// Mitsubishi GX Works2 project: PID_slave_test1   PLC: FX3U/FX3UC

// global labels: Global1
VAR_GLOBAL
  lampe_0 AT Y000 : BOOL;
  lampe_1 AT Y001 : BOOL;
  lampeVar_0 AT M100 : BOOL;
  lampeVar_1 AT M101 : BOOL;
  anaDig AT D8260 : INT;
  digAna AT D8262 : INT;
  slider AT D0 : INT;
  tank AT D1 : INT;
  Output_PID AT D40 : INT;  (* Utgangs signal sendt ut fra PID *)
  Input_Referance AT D42 : INT;  (* Referanse verdi sendt til PID *)
  Input_Process AT D44 : INT;  (* Prosess verdi Sendt til PID *)
  Input_ManualValue AT D54 : INT;  (* Manuell verdi sendt til PID *)
  Input_ManualMode AT M105 : BOOL;  (* Valg av Manuell "1" eller Auto "0" *)
  Input_SamplingsTime AT D56 : INT;  (* Samplingstid sendt til PID *)
  Input_OperationModus AT M106 : BOOL;  (* Valg av direkte "1" eller Revers "0" Regulering *)
  Inpud_IntegratorModus AT M107 : BOOL;  (* Valg av Integrator virkning på regulator *)
  Input_NomValue AT D58 : INT;  (* Nominelt pådrag *)
  Input_DerivatorModus AT M108 : BOOL;  (* Valg av Derivator virkning på regulator *)
  Input_MaxPådrag AT D60 : INT;  (* Max pådrag *)
  Input_MinPådrag AT D62 : INT;  (* Min pådrag *)
END_VAR

// task Task_01 (event TRUE, interval 0, priority 31): POU_01

PROGRAM POU_01
VAR
  TestBlock_1 : TestBlock;
  tiss_1 : tiss;
  TestBlock_2 : TestBlock;
  tiss_2 : tiss;
  tiss_3 : tiss;
END_VAR
(* structured ladder/FBD written out as ST: instructions are called as NAME(EN, inputs, outputs); _pN, _eN, _tN stand for wires *)
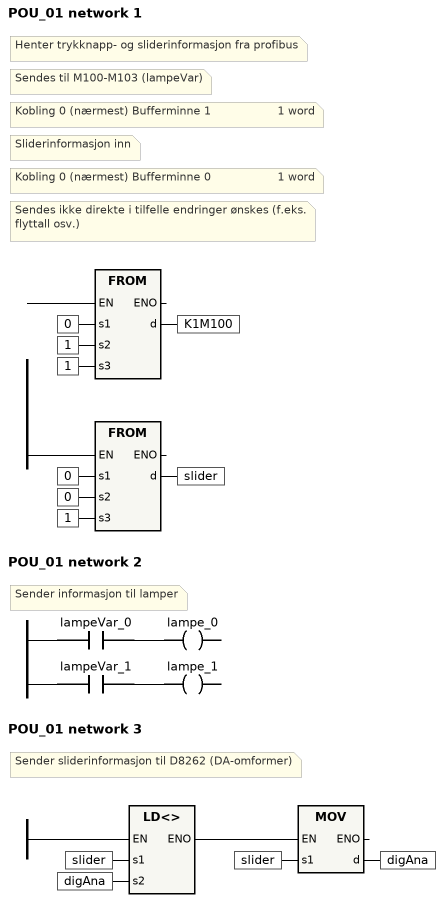
(* network 1 *)
(* Henter trykknapp- og sliderinformasjon fra profibus *)
(* Sendes til M100-M103 (lampeVar) *)
(* Kobling 0 (nærmest) Bufferminne 1                   1 word *)
(* Sliderinformasjon inn *)
(* Kobling 0 (nærmest) Bufferminne 0                   1 word *)
(* Sendes ikke direkte i tilfelle endringer ønskes (f.eks. flyttall osv.) *)
FROM(TRUE, 0, 1, 1, K1M100);
FROM(TRUE, 0, 0, 1, slider);
(* network 2 *)
(* Sender informasjon til lamper *)
lampe_0 := lampeVar_0;
lampe_1 := lampeVar_1;
(* network 3 *)
(* Sender sliderinformasjon til D8262 (DA-omformer) *)
_e1 := LD<>(TRUE, slider, digAna);
MOV(_e1, slider, digAna);
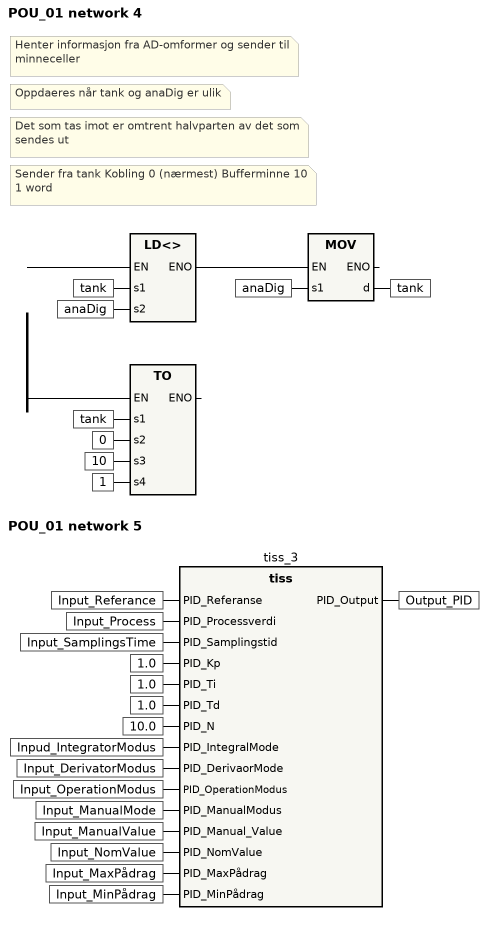
(* network 4 *)
(* Henter informasjon fra AD-omformer og sender til minneceller *)
(* Oppdaeres når tank og anaDig er ulik *)
(* Det som tas imot er omtrent halvparten av det som sendes ut *)
(* Sender fra tank Kobling 0 (nærmest) Bufferminne 10           1 word *)
_e1 := LD<>(TRUE, tank, anaDig);
MOV(_e1, anaDig, tank);
TO(TRUE, tank, 0, 10, 1);
(* network 5 *)
tiss_3(PID_Referanse := Input_Referance, PID_Processverdi := Input_Process, PID_Samplingstid := Input_SamplingsTime, PID_Kp := 1.0, PID_Ti := 1.0, PID_Td := 1.0, PID_N := 10.0, PID_IntegralMode := Inpud_IntegratorModus, PID_DerivaorMode := Input_DerivatorModus, PID_OperationModus := Input_OperationModus, PID_ManualModus := Input_ManualMode, PID_Manual_Value := Input_ManualValue, PID_NomValue := Input_NomValue, PID_MaxPådrag := Input_MaxPådrag, PID_MinPådrag := Input_MinPådrag, PID_Output => Output_PID);
END_PROGRAM

FUNCTION_BLOCK TestBlock
VAR_INPUT
  PID_Referanse : INT;  (* Referanseverdi PID blokk *)
  PID_Processverdi : INT;  (* Prosessverdi PID blokk *)
  PID_Samplingstid : REAL;  (* Samplingstid PID blokk (ms) *)
  PID_Kp : REAL;  (* KP PID blokk *)
  PID_Ti : REAL;  (* Ti PID blokk *)
  PID_Td : REAL;  (* Td PID blokk *)
  PID_N : REAL;  (* Filter konstant for Tf *)
  PID_IntegralMode : BOOL;  (* Integrator for PID blokk *)
  PID_DerivaorMode : BOOL;  (* Derivator for PID blokk *)
  PID_OperationModus : BOOL;  (* Framover kobling "0", bakoverkobling "1" *)
  PID_ManualModus : BOOL;  (* Auto "0" , Manuell pådrag "1" *)
END_VAR
VAR
  PID_Mellomregning_TN_F : REAL;  (* Mellomregning for T*N *)
  PID_Alpha : REAL;  (* Beregnet alpha verdi *)
  PID_ErrorValue_W : INT;  (* Beregnet error verdi *)
  PID_ErrorValue_F : ARRAY [0..1] OF REAL;  (* Beregnet error verdi *)
  PID_PGain : ARRAY [0..1] OF REAL;  (* Beregnet P forsterkning (Denne og forrige verdi) *)
  PID_Skalert_Processverdi_DW : DWORD;  (* Process verdi skalert med en faktor 2 *)
  PID_Skalert_Processverdi_W : WORD;  (* Process verdi skalert med en faktor 2 *)
  PID_Beta : REAL;  (* Beregnet alpha verdi *)
  PID_Mellomregning_TNplusTd_F : REAL;  (* Mellom regning for T*N+Td *)
  PID_Mellomregning_Integrator : REAL;  (* Mellom regning Kp*alpha*error[0] *)
  PID_IGain : ARRAY [0..1] OF REAL;  (* Beregnet I forsterkning (Denne og forrige verdi) *)
  PID_Mellomregning_Derivator : REAL;  (* Mellom regning for (Kp*Td/T)*(1-beta) *)
  PID_DGain : ARRAY [0..1] OF REAL;  (* Beregnet D forsterkning (Denne og forrige verdi) *)
  PID_Skalert_Processverdi_F : ARRAY [0..1] OF REAL;  (* Process verdi skalert med en faktor 2 *)
  PID_Gain : REAL;  (* Beregnet sum av pådrag *)
END_VAR
VAR_OUTPUT
  PID_Output : REAL;  (* Utgangsverdi fra PID-reg *)
END_VAR
(* structured ladder/FBD written out as ST: instructions are called as NAME(EN, inputs, outputs); _pN, _eN, _tN stand for wires *)
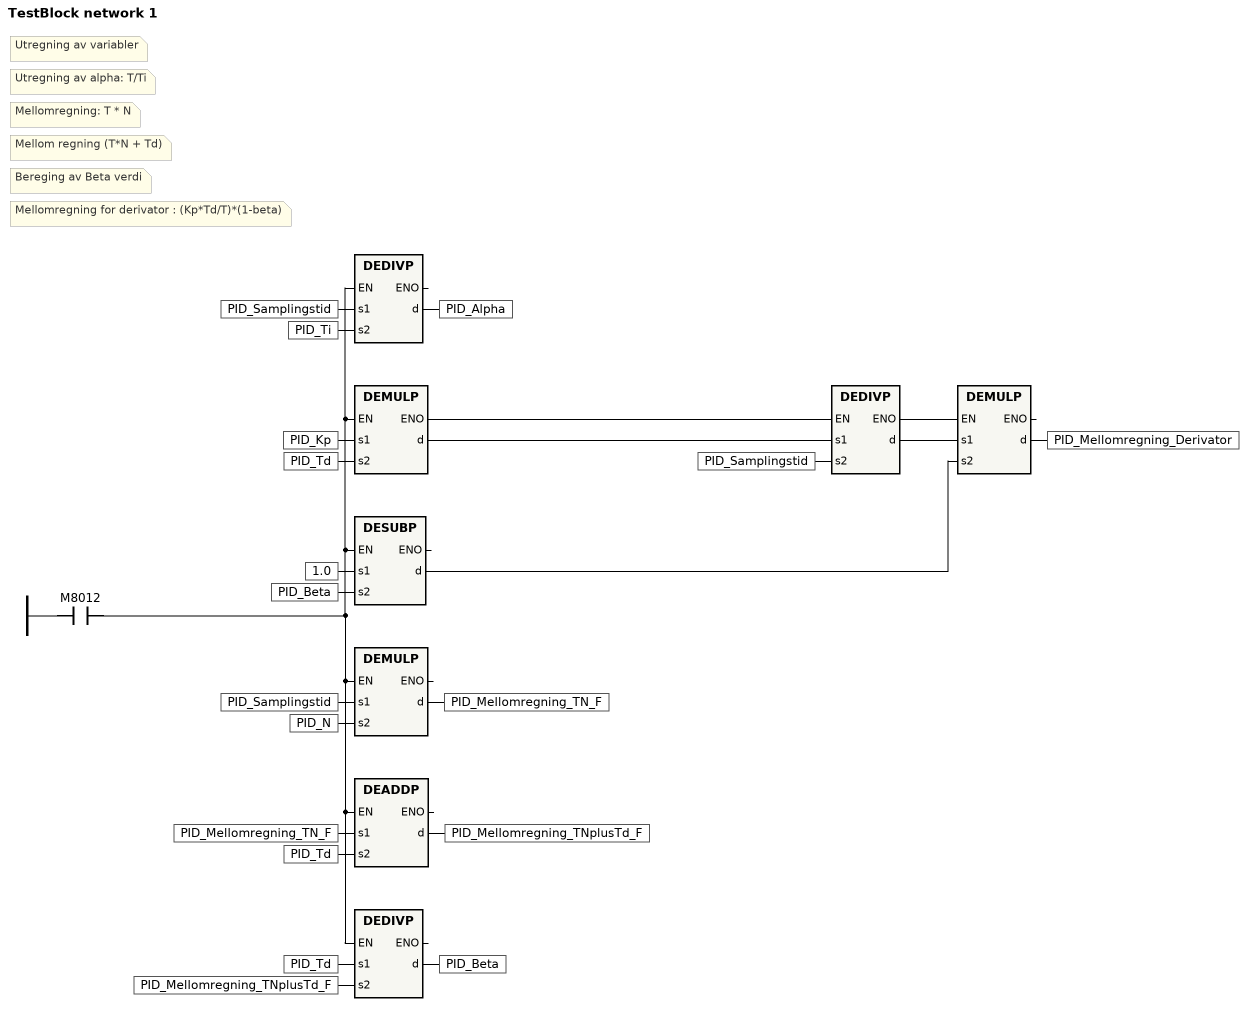
(* network 1 *)
(* Utregning av variabler *)
(* Utregning av alpha: T/Ti *)
(* Mellomregning: T * N *)
(* Mellom regning (T*N + Td) *)
(* Bereging av Beta verdi *)
(* Mellomregning for derivator : (Kp*Td/T)*(1-beta) *)
DEDIVP(M8012, PID_Samplingstid, PID_Ti, PID_Alpha);
DEMULP(M8012, PID_Samplingstid, PID_N, PID_Mellomregning_TN_F);
DEADDP(M8012, PID_Mellomregning_TN_F, PID_Td, PID_Mellomregning_TNplusTd_F);
DEDIVP(M8012, PID_Td, PID_Mellomregning_TNplusTd_F, PID_Beta);
_e2 := DEMULP(M8012, PID_Kp, PID_Td, _t1);
_e4 := DEDIVP(_e2, _t1, PID_Samplingstid, _t3);
DESUBP(M8012, 1.0, PID_Beta, _t5);
DEMULP(_e4, _t3, _t5, PID_Mellomregning_Derivator);
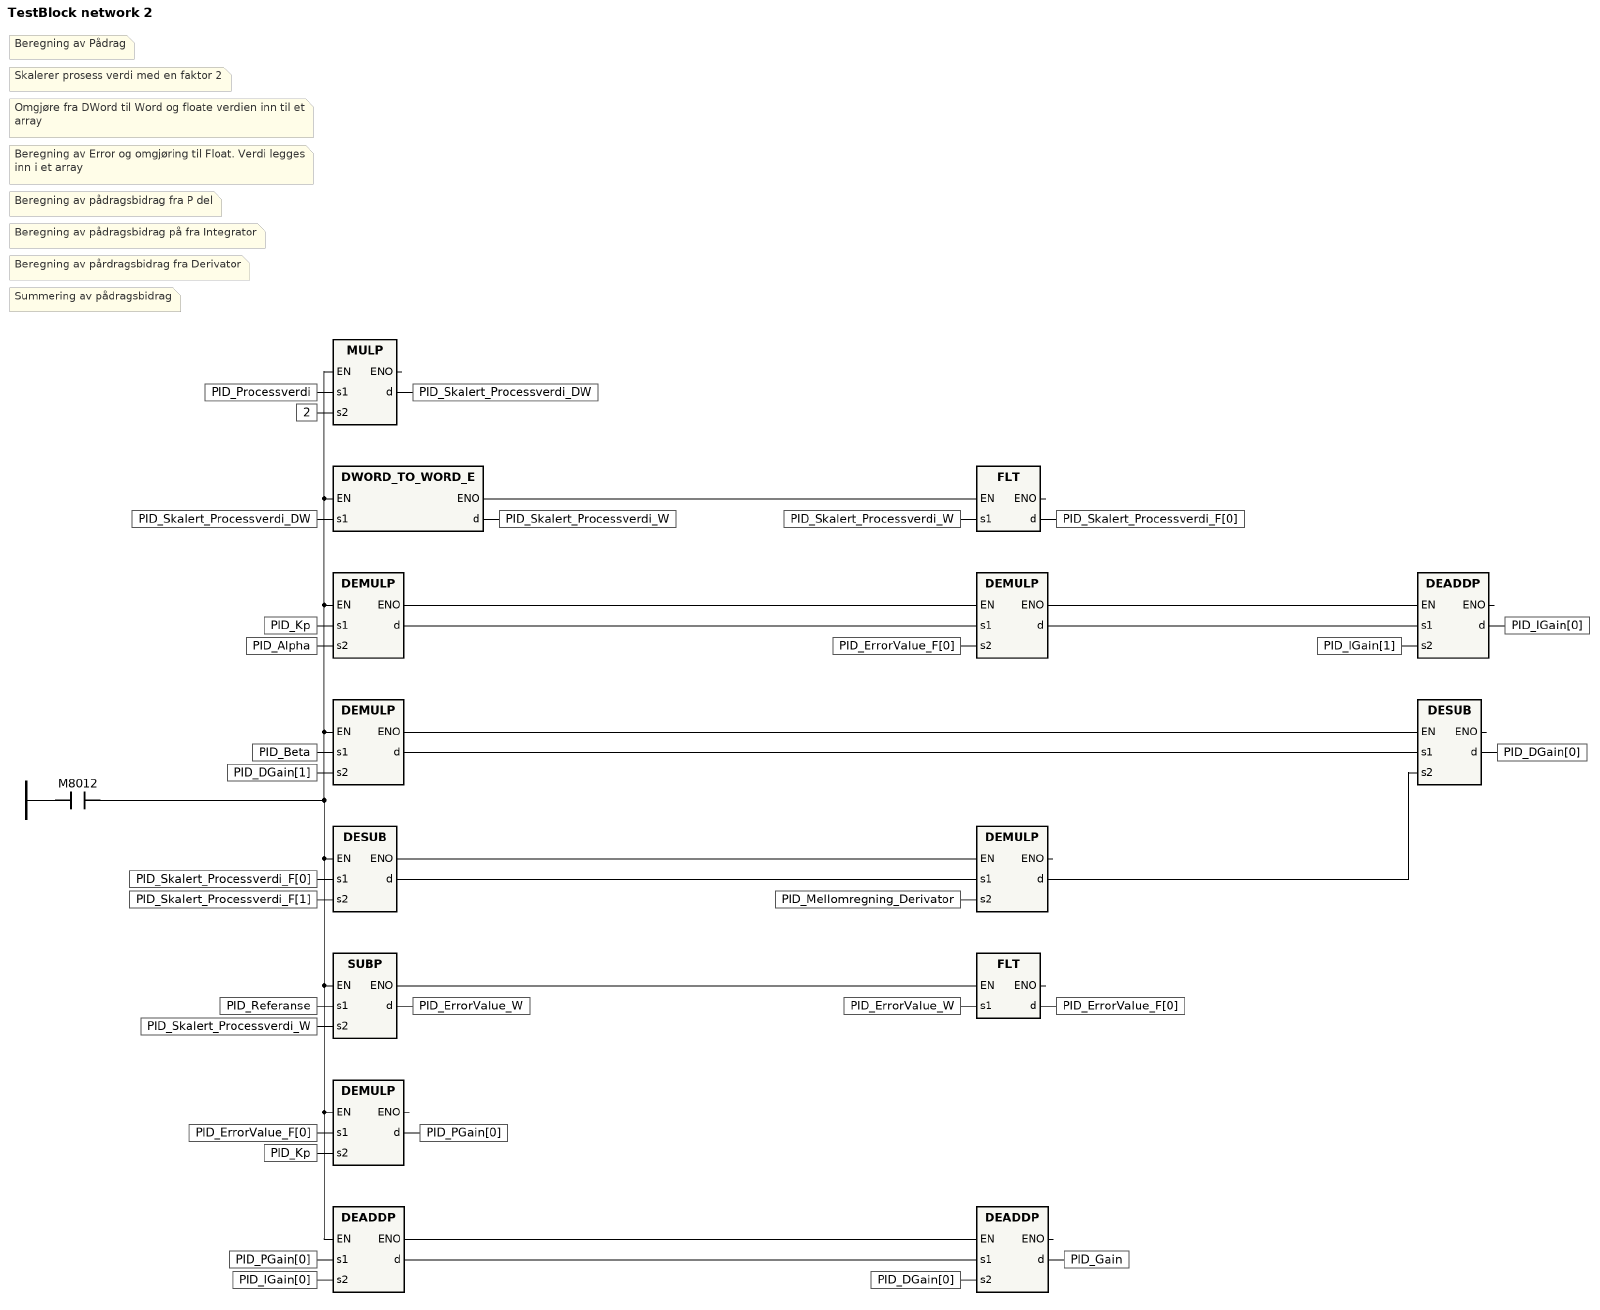
(* network 2 *)
(* Beregning av Pådrag *)
(* Skalerer prosess verdi med en faktor 2 *)
(* Omgjøre fra DWord til Word og floate verdien inn til et array *)
(* Beregning av Error og omgjøring til Float. Verdi legges inn i et array *)
(* Beregning av pådragsbidrag fra P del *)
(* Beregning av pådragsbidrag på fra Integrator *)
(* Beregning av pårdragsbidrag fra Derivator *)
(* Summering av pådragsbidrag *)
MULP(M8012, PID_Processverdi, 2, PID_Skalert_Processverdi_DW);
_e1 := DWORD_TO_WORD_E(M8012, PID_Skalert_Processverdi_DW, PID_Skalert_Processverdi_W);
FLT(_e1, PID_Skalert_Processverdi_W, PID_Skalert_Processverdi_F[0]);
_e2 := SUBP(M8012, PID_Referanse, PID_Skalert_Processverdi_W, PID_ErrorValue_W);
FLT(_e2, PID_ErrorValue_W, PID_ErrorValue_F[0]);
DEMULP(M8012, PID_ErrorValue_F[0], PID_Kp, PID_PGain[0]);
_e4 := DEMULP(M8012, PID_Kp, PID_Alpha, _t3);
_e6 := DEMULP(_e4, _t3, PID_ErrorValue_F[0], _t5);
DEADDP(_e6, _t5, PID_IGain[1], PID_IGain[0]);
_e8 := DEMULP(M8012, PID_Beta, PID_DGain[1], _t7);
_e10 := DESUB(M8012, PID_Skalert_Processverdi_F[0], PID_Skalert_Processverdi_F[1], _t9);
DEMULP(_e10, _t9, PID_Mellomregning_Derivator, _t11);
DESUB(_e8, _t7, _t11, PID_DGain[0]);
_e13 := DEADDP(M8012, PID_PGain[0], PID_IGain[0], _t12);
DEADDP(_e13, _t12, PID_DGain[0], PID_Gain);
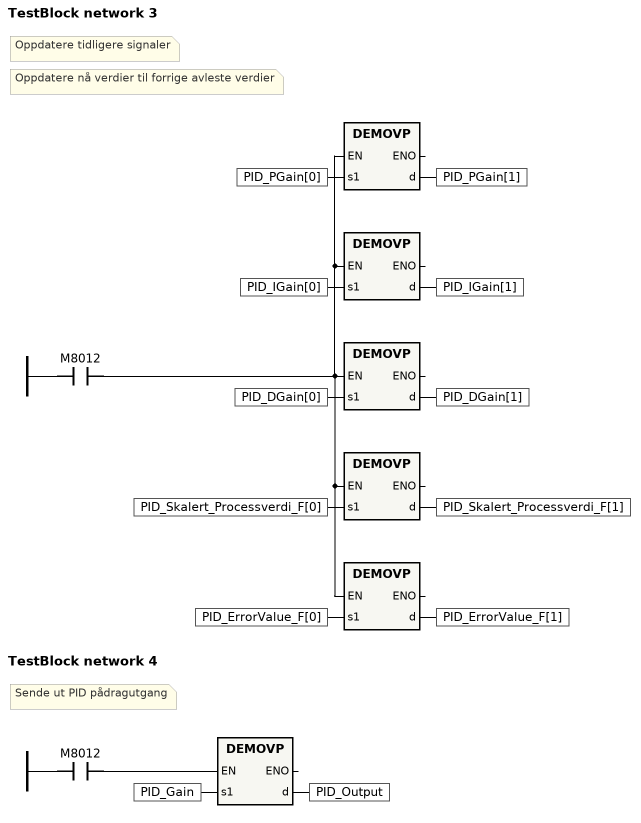
(* network 3 *)
(* Oppdatere tidligere signaler *)
(* Oppdatere nå verdier til forrige avleste verdier *)
DEMOVP(M8012, PID_PGain[0], PID_PGain[1]);
DEMOVP(M8012, PID_IGain[0], PID_IGain[1]);
DEMOVP(M8012, PID_DGain[0], PID_DGain[1]);
DEMOVP(M8012, PID_Skalert_Processverdi_F[0], PID_Skalert_Processverdi_F[1]);
DEMOVP(M8012, PID_ErrorValue_F[0], PID_ErrorValue_F[1]);
(* network 4 *)
(* Sende ut PID pådragutgang *)
DEMOVP(M8012, PID_Gain, PID_Output);
END_FUNCTION_BLOCK

FUNCTION_BLOCK tiss
VAR_INPUT
  PID_Referanse : INT;  (* Referanseverdi PID blokk *)
  PID_Processverdi : INT;  (* Prosessverdi PID blokk *)
  PID_Samplingstid : INT;  (* Samplingstid PID blokk (ms) *)
  PID_Kp : REAL;  (* KP PID blokk *)
  PID_Ti : REAL;  (* Ti PID blokk *)
  PID_Td : REAL;  (* Td PID blokk *)
  PID_N : REAL;  (* Filter konstant for Tf *)
  PID_IntegralMode : BOOL;  (* Integrator for PID blokk *)
  PID_DerivaorMode : BOOL;  (* Derivator for PID blokks *)
  PID_OperationModus : BOOL;  (* Direkte kobling "1", reversert "0" *)
  PID_ManualModus : BOOL;  (* Auto "0" , Manuell pådrag "1" *)
END_VAR
VAR
  PID_Alpha : REAL;  (* Beregnet alpha verdi *)
  PID_Beta : REAL;  (* Beregnet alpha verdi *)
END_VAR
VAR_INPUT
  PID_Manual_Value : INT;  (* Manuelt pådrag verdi *)
  PID_NomValue : INT;  (* Nominelt pådrags verdi *)
END_VAR
VAR_OUTPUT
  PID_Output : INT;  (* Utgangsverdi fra PID-reg *)
END_VAR
VAR_INPUT
  PID_MaxPådrag : INT;  (* Max pådrags verdi *)
  PID_MinPådrag : INT;  (* Min pådrags verdi *)
END_VAR
VAR
  PID_ErrorValue_F : ARRAY [0..1] OF REAL;  (* Beregnet error verdi *)
  PID_PGain : ARRAY [0..1] OF REAL;  (* Beregnet P forsterkning (Denne og forrige verdi) *)
  PID_IGain : ARRAY [0..1] OF REAL;  (* Beregnet I forsterkning (Denne og forrige verdi) *)
  PID_DGain : ARRAY [0..1] OF REAL;  (* Beregnet D forsterkning (Denne og forrige verdi) *)
  PID_Gain : REAL;  (* Beregnet sum av pådrag *)
  PID_Mellomregning_Samplingstid : REAL;  (* Mellomregning av samplingstid *)
  PID_Mellomregning_NomVal : REAL;  (* Mellomregning av nominelt pådrag *)
  PID_Skalert_Processverdi_F : ARRAY [0..1] OF REAL;  (* Process verdi skalert med en faktor 2 *)
  PID_Skalert_Samplingstid : REAL;  (* Skalert samplingstid i sekunder *)
  PID_Referanse_F : REAL;  (* Referanse verdi i Float *)
  PID_Skalert_NomVal : REAL;  (* Nominelt pådrag i bits *)
  PID_Mellomregning_MaxVal : REAL;  (* Mellomregning av max pådrag *)
  PID_Mellomregning_MinVal : REAL;  (* Mellomregning av min pådrag *)
  PID_Skalert_MaxVal : REAL;  (* Max pådrag i bits *)
  PID_Skalert_MinVal : REAL;  (* Min pådrag i bits *)
  PID_Mellomregning_ManuellVal : REAL;  (* Mellomregning av manuelt pådrag *)
  PID_Skalert_ManVal : REAL;  (* Manuelt pådrag i bits *)
END_VAR
(*Omgjøring av samplingstid fra ms til s*)
FLT(TRUE , PID_Samplingstid, PID_Mellomregning_Samplingstid);
PID_Skalert_Samplingstid := PID_Mellomregning_Samplingstid/1000.0;

(*Timer for samplingstid*)
OUT_T(NOT(TS200), TC200, PID_Samplingstid/10);

(*Systemet vil gå inn i koden hvert samplingstid som er satt*)
IF TS200 THEN	
	
	(*Regning av konstanter alpha, beta og omgjøring av prosess, nominelt-, min og max pådrag og ref verdi til float*)
	PID_Alpha := PID_Skalert_Samplingstid/PID_Ti;
	PID_Beta := PID_Td/(PID_Td + (PID_Skalert_Samplingstid*pid_n));
	FLT(TRUE,PID_Referanse, PID_Referanse_F);
	FLT(TRUE,PID_Processverdi*2,PID_Skalert_Processverdi_F[0]);
	FLT(TRUE, PID_NomValue, PID_Mellomregning_NomVal);
	FLT(TRUE, PID_MaxPådrag, PID_Mellomregning_MaxVal);
	FLT(TRUE, PID_MinPådrag, PID_Mellomregning_MinVal);
	FLT(TRUE, PID_Manual_Value, PID_Mellomregning_ManuellVal);
	
	
	
	(*Skalering av nominelt, max og min pådrag til bits*)
	PId_Skalert_NomVal := PID_Mellomregning_NomVal*40.79;
	PID_Skalert_MaxVal:= PID_Mellomregning_MaxVal*40.79;
	PID_Skalert_MinVal:= PID_Mellomregning_MinVal*40.79;
	PID_Skalert_ManVal:= PID_Mellomregning_ManuellVal*40.79;
	
	(*Regning av avvik mtp om det er direkte eller revers regulering*)
	IF PID_OperationModus THEN
		PID_ErrorValue_F[0] := PID_Skalert_Processverdi_F[0] - PID_Referanse_F;
	ELSE
		PID_ErrorValue_F[0] := PID_Referanse_F - PID_Skalert_Processverdi_F[0];
	END_IF;
	
	(*PID regulering, enten manuell eller auto modus*)
	IF PID_ManualModus THEN 
		INT(TRUE, PID_Skalert_ManVal, PID_Output);
	ELSE 
		PID_PGain[0] := PID_Kp*(PID_ErrorValue_F[0]-PID_ErrorValue_F[1]);
		IF PID_IntegralMode THEN
			PID_IGain[0] := PID_Kp*PID_Alpha*PID_ErrorValue_F[0];
		ELSE
			PID_IGain[0] := 0.0;
		END_IF;
		IF PID_DerivaorMode THEN
			PID_DGain[0] := (PID_Beta*PID_DGain[1]) - ((PID_Kp*PID_Td/PID_Skalert_Samplingstid)*(1.0-PID_Beta)*(PID_Skalert_Processverdi_F[0]-PID_Skalert_Processverdi_F[1]));
		ELSE 
			PID_DGain[0] := 0.0;
		END_IF;
		PID_Gain := PID_PGain[0] + PID_IGain[0] + PID_DGain[0] + PId_Skalert_NomVal;
		
			(*Oppdatering av verdier*)
		PID_ErrorValue_F[1] := PID_ErrorValue_F[0];
		PID_Skalert_Processverdi_F[1] := PID_Skalert_Processverdi_F[0];
		PID_PGain[1] := PID_PGain[0];
		PID_IGain[1] := PID_IGain[0];
		PID_DGain[1] := PID_DGain[0];
	
		
		IF PID_Gain > PID_Skalert_MaxVal THEN
			PID_Gain:= PID_Skalert_MaxVal;
		ELSIF PID_Gain < PID_Skalert_MinVal THEN 
			PID_Gain:= PID_Skalert_MinVal;
		ELSE
			PID_Gain:= PID_Gain;
		END_IF;
		
		(*Utgang fra PID regulator*)
		INT(TRUE , PID_Gain, PID_Output);
	END_IF;
	
	
	
	

	
	
	
ELSE
;
END_IF;
END_FUNCTION_BLOCK
